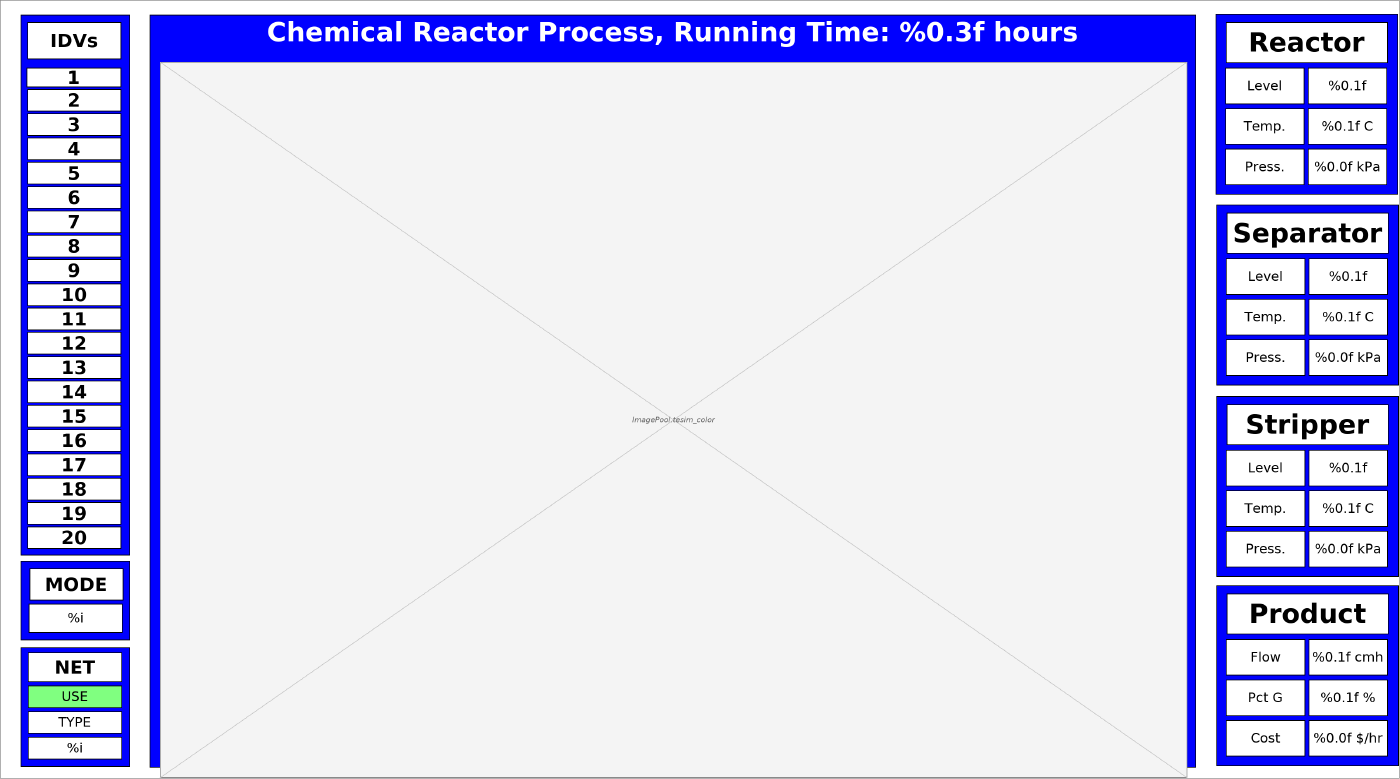
VISUALIZATION TankView  // 1899x1058
    Rectangle (203,20 1419x1022), "Chemical Reactor Process, Running Time: %0.3f hours", text variable: OPTIME
    Rectangle (1649,19 247x245)
    Rectangle (1663,30 219x55), "Reactor"
    Rectangle (1774,92 107x49), "%0.1f", text variable: G_IO.XMEAS[8]
    Rectangle (1774,147 107x49), "%0.1f C", text variable: G_IO.XMEAS[9]
    Rectangle (1774,202 107x49), "%0.0f kPa", text variable: G_IO.XMEAS[7]
    Rectangle (1662,92 107x49), "Level"
    Rectangle (1662,147 107x49), "Temp."
    Rectangle (1662,202 107x49), "Press."
    Rectangle (1650,278 247x245)
    Rectangle (1664,289 219x55), "Separator"
    Rectangle (1775,351 107x49), "%0.1f", text variable: G_IO.XMEAS[12]
    Rectangle (1775,406 107x49), "%0.1f C", text variable: G_IO.XMEAS[11]
    Rectangle (1775,461 107x49), "%0.0f kPa", text variable: G_IO.XMEAS[13]
    Rectangle (1663,351 107x49), "Level"
    Rectangle (1663,406 107x49), "Temp."
    Rectangle (1663,461 107x49), "Press."
    Rectangle (1650,538 247x245)
    Rectangle (1664,549 219x55), "Stripper"
    Rectangle (1775,611 107x49), "%0.1f", text variable: G_IO.XMEAS[15]
    Rectangle (1775,666 107x49), "%0.1f C", text variable: G_IO.XMEAS[18]
    Rectangle (1775,721 107x49), "%0.0f kPa", text variable: G_IO.XMEAS[16]
    Rectangle (1663,611 107x49), "Level"
    Rectangle (1663,666 107x49), "Temp."
    Rectangle (1663,721 107x49), "Press."
    Rectangle (1650,795 247x245)
    Rectangle (1664,806 219x55), "Product"
    Rectangle (1775,868 107x49), "%0.1f cmh", text variable: G_IO.XMEAS[17]
    Rectangle (1775,923 107x49), "%0.1f %", text variable: G_IO.XMEAS[40]
    Rectangle (1775,978 107x49), "%0.0f $/hr", text variable: G_IO.COST
    Rectangle (1663,868 107x49), "Flow"
    Rectangle (1663,923 107x49), "Pct G"
    Rectangle (1663,978 107x49), "Cost"
    Rectangle (221,200 190x49), "%0.3f kscmh", text variable: G_IO.XMEAS[1]
    Rectangle (221,364 192x49), "%0.1f kgph", text variable: G_IO.XMEAS[2]
    Rectangle (221,515 202x49), "%0.1f kgph", text variable: G_IO.XMEAS[3]
    Rectangle (460,915 200x49), "%0.3f kscmh", text variable: G_IO.XMEAS[4]
    Rectangle (28,20 148x734)
    Rectangle (37,30 127x50), "IDVs"
    Rectangle (36,92 128x26), "1", invisible if: Not(udint_to_bool(IDV[1]))
    Rectangle (37,121 127x30), "2", invisible if: Not(udint_to_bool(IDV[2]))
    Rectangle (37,154 127x30), "3", invisible if: Not(udint_to_bool(IDV[3]))
    Rectangle (37,187 127x30), "4", invisible if: Not(udint_to_bool(IDV[4]))
    Rectangle (37,220 127x30), "5", invisible if: Not(udint_to_bool(IDV[5]))
    Rectangle (37,253 127x30), "6", invisible if: Not(udint_to_bool(IDV[6]))
    Rectangle (37,286 127x30), "7", invisible if: Not(udint_to_bool(IDV[7]))
    Rectangle (37,319 127x30), "8", invisible if: Not(udint_to_bool(IDV[8]))
    Rectangle (37,352 127x30), "9", invisible if: Not(udint_to_bool(IDV[9]))
    Rectangle (37,385 127x30), "10", invisible if: Not(udint_to_bool(IDV[10]))
    Rectangle (37,418 127x30), "11", invisible if: Not(udint_to_bool(IDV[11]))
    Rectangle (37,451 127x30), "12", invisible if: Not(udint_to_bool(IDV[12]))
    Rectangle (37,484 127x30), "13", invisible if: Not(udint_to_bool(IDV[13]))
    Rectangle (37,517 127x30), "14", invisible if: Not(udint_to_bool(IDV[14]))
    Rectangle (37,550 127x30), "15", invisible if: Not(udint_to_bool(IDV[15]))
    Rectangle (37,583 127x30), "16", invisible if: Not(udint_to_bool(IDV[16]))
    Rectangle (37,616 127x30), "17", invisible if: Not(udint_to_bool(IDV[17]))
    Rectangle (37,649 127x30), "18", invisible if: Not(udint_to_bool(IDV[18]))
    Rectangle (37,682 127x30), "19", invisible if: Not(udint_to_bool(IDV[19]))
    Rectangle (37,715 127x30), "20", invisible if: Not(udint_to_bool(G_IO.IDV[20]))
    Rectangle (28,879 148x162)
    Rectangle (38,886 127x40), "NET"
    Rectangle (38,1001 127x30), "%i", text variable: NET_TYPE
    Rectangle (38,931 127x30), "USE", invisible if: Not(GO)
    Rectangle (38,966 127x30), "TYPE"
    Rectangle (28,762 148x107)
    Rectangle (40,772 127x43), "MODE"
    Rectangle (39,820 127x39), "%i", text variable: MODE
    Image (217,84 1393x972), image: ImagePool.tesim_color
END_VISUALIZATION

(* stored: Version 1.1.0.1, ProductVersion 3.1.4020.12
   Visu TankView: Id {f4f04a74-56cf-403a-ae2f-59b885671ef0} *)
